Universal Robots PolyScope program: v001_robot_to_HALCON.urp

Program v001_robot_to_HALCON (installation=default directory=/programs createdIn=3.0.17779.0 lastSavedIn=5.9.1.1031110 robotSerialNumber=20195501059)
Calibrated DH parameters: a=[0.000146, -0.418764, -0.053981, 0.000058, -0.000023, 0]; d=[0.162545, 37.319448, -206.067439, 168.881546, 0.09955, 0.099464]; alpha=[1.57004, -0.001979, 0.002304, 1.570607, -1.57066, 0]; deltaTheta=[0, -0.174616, -1.258233, 1.432844, -0.000001, 0]
Robot Program (runOnlyOnce=true)
  MoveJ speed 60 deg/s, acceleration 80 deg/s^2 (useActiveTCP=true) feature=Base
    Waypoint Waypoint_1: TCP in base x=127.32 y=-316.711 z=182.361 mm, rx=-0.9513 ry=-2.7955 rz=0.1885 rad; joints [99.464, -110.447, 127.368, -108.398, 257.399, 46.878] deg; TCP offset x=0 y=0 z=174 mm, rx=0 ry=0 rz=0 rad
  Call vision_connect
  Loop Counting (count=5) loopVariable(name=Loop_2)
    MoveL speed 250 mm/s, acceleration 1200 mm/s^2 (useActiveTCP=true) feature=Base
      Waypoint Waypoint_2: TCP in base x=127.334 y=-409.734 z=182.348 mm, rx=-0.9512 ry=-2.7955 rz=0.1884 rad; joints [97.344, -97.173, 117.846, -112.619, 257.445, 44.715] deg
    Call vision_find
    MoveL speed 250 mm/s, acceleration 1200 mm/s^2 (useActiveTCP=true) feature=Base
      Waypoint Waypoint_1: TCP in base x=127.32 y=-316.711 z=182.361 mm, rx=-0.9513 ry=-2.7955 rz=0.1885 rad; joints [99.464, -110.447, 127.368, -108.398, 257.399, 46.878] deg
  Call vision_disconnect
SubProgram -> vision_connect
SubProgram -> vision_disconnect
SubProgram -> vision_find
SubProgram vision_connect (keepSynchronizedWithDisk=false) programFile=/programs/vision_connect.urp
  v_connected := False
  Loop While (checkContinuously=false) expression=v_connected≟ False
    v_connected := socket_open("192.168.0.251",3000,"socket0")
    Wait Sleep waitTime=0.2
    Script: TargetObject = [0,0,0,0,0,0]
SubProgram vision_find (keepSynchronizedWithDisk=false) programFile=/programs/vision_find.urp
  Script: socket_send_line("r","socket0")
  TargetObject := [0,0,0,0,0,0]
  Loop While (checkContinuously=false) expression=TargetObject[0]≟0
    TargetObject := socket_read_ascii_float(5,"socket0")
    Wait Sleep waitTime=0.1
  Vcommand_idx := TargetObject[1]
  TargetX := TargetObject[2]
  TargetY := TargetObject[3]
  TargetRotation := -d2r(TargetObject[4])
  TargetPercent := TargetObject[5]
SubProgram vision_disconnect (keepSynchronizedWithDisk=false) programFile=/programs/vision_disconnect.urp
  v_connected := False
  Script: socket_close("socket0")
